TYPE HMIWindowSwitch :
STRUCT
	MinPage	:	INT;
	MaxPage	:	INT;
	SelectedPage	:	INT;
	SelectedTab	:	STRING;
	NextPageIsEnabled	:	BOOL;
	NextPageIsPressed	:	BOOL;
	PreviousPageIsEnabled	:	BOOL;
	PreviousPageIsPressed	:	BOOL;
END_STRUCT
END_TYPE

(* stored: Version 1.1.0.1
   DUT HMIWindowSwitch: Id {38d5fac8-6f53-4907-b1d4-0d1bdb22b7b8} *)
